Staubli VAL3: sad_proj_sin.pjx

--- sad_proj_sin.pjx ---
Parameters version=s7.7.1 stackSize=5000 millimeterUnit=true
Program file=check_cmt.pgx
Program file=motion_cntl.pgx
Program file=open_socket.pgx
Program file=read_data.pgx
Program file=send_data.pgx
Program file=show_data.pgx
Program file=start.pgx
Program file=stop.pgx
Data file=sad_proj_sin.dtx

--- check_cmt.pgx ---
public program check_cmt()
  local num sCheck
  local num nEOS
begin

  clearBuffer(sioASCII)

  nEOS = 0
  sCheck = sioSet(sioASCII,nEOS)
  sCheck = sioSet(sioASCII,13)

  if sCheck == 1
    putln("Communication is OK !")
    check_status = true
  elseIf sCheck != 1
    putln("Communication error !")
    check_status = false
  endIf

end

--- init_prgm.pgx ---
public program init_prgm()
begin

  // mise en rotation pompe vitesse nulle
    aioSet(Tpompe,0)
    put("Pompe en rotation")
    // arrêt pompe
    dioSet(doPompe,0)
    put("Pompe arret")
    // fermeture obturateur
    dioSet(doValve2,0)
    dioSet(doValve1,1)
    put("Obturateur fermé")

end

--- launch_print.pgx ---
program launch_print()
begin

  // ouverture obturateur
    dioSet(doValve1,0)
    dioSet(doValve2,1)
    put("Obturateur ouvert")
    delay(2)
    // mise en marche pompe vitesse faible
    dioSet(doPompe,1)
    put("Pompe en marche")
    delay(2)
    // mise en rotation pompe vitesse donnée
    aioSet(Tpompe,1.2)
    put("Pompe en rotation")

end

--- read_ID.pgx ---
public program read_ID()
  local bool non_stop
begin

  non_stop = true

  do

    putln(getMoveId())
    putln(getMonitorSpeed())

  until non_stop != true

end

--- show_data.pgx ---
public program show_data()
begin

   do
    cls()
    put("Reference Velocity [mm/s]: ")
    put(Ref_Vel)
    putln("")
    //cls()
    put("Robot Velocity [mm/s]: ")
    put(getSpeed(tTool))
    putln("")
    //cls()
    put("Error (Ref-Rob) [mm/s]: ")
    put(Ref_Vel - getSpeed(tTool))
    putln("")
    //cls()
    put("Current position: ")
    put(getMoveId())
    putln("")


    delay(0.001)
    //putln("")
  until check_status != true

end
